Omron Sysmac Studio project BPP_17003_21Fev2018_13h32 (Sysmac Studio 1.21.1.6, StandardProject)

# Controller new_Controller_0: NJ101-1020 version 1.13
Units and slaves: Node10 : GX-JC06(IN,X2,X3) Main device (E001); Node11 : Inverter i550 Cabinet (E002); Node12 : Inverter i550 Cabinet (E003); Node13 : Inverter i550 Cabinet (E004); Node14 : Inverter i550 Cabinet (E005); Node15 : Inverter i550 Cabinet (E006); Node16 : Inverter i550 Cabinet (E007); Node21 : Inverter i550 Cabinet (E008); Node22 : Inverter i550 Cabinet (E009); Node23 : Inverter i550 Cabinet (E010); Node24 : Inverter i550 Cabinet (E011); Node25 : Inverter i550 Cabinet (E012); Node26 : Inverter i550 Cabinet (E013); Node30 : GX-JC06(X4,X5,X6) Sub-device (E014); Power Supply : NJ-Px3001; CPU : NJ101-1020; 0 [Unit 1] : CJ1W-ECT21 (J01); 1 [Unit 2] : CJ1W-EIP21 (J02); 2 : CJ1W-ID262 (J03); 3 : CJ1W-ID262 (J04); 4 : CJ1W-OD262 (J05); 5 : CJ1W-OD212 (J06)
Axis MC_Axis320M1, settings changed from default: AxisType=ServoType, UnitsConversion=EnumElement2, UnitsNumerator=8388608, UnitsDenominator=120, MaxVelocity=1000, StartVelocity=1000, MaxJogVelocity=100, MaxAcceleration=10, MaxDeceleration=10, WarningTorqueLimitPositive=90, WarningTorqueLimitNegative=90, HomingMode=BackupAndPressingTime, StartDirection=NegativeDirection, HomingVelocity=50, HomingApproachVelocity=10, HomingAcceleration=10, CompensationVelocity=10, EncoderTypes=Abs
Task PrimaryTask (priority 4, period or condition 2000): Programa

TYPE DataMotor : STRUCT
    Auto : BOOL;  (* Equipamento em Automatico *)
    Alarm : BOOL;  (* Equipamento em Alarme *)
    FcaFwd : BOOL;  (* Comando automatico Avanço *)
    FcaRev : BOOL;  (* Comando automatico Recuo *)
    FeFwd : BOOL;  (* Encravamento Avanço - Não pode Executar *)
    FeRev : BOOL;  (* Encravamento Recuo - Não pode Executar *)
    OutFwd : BOOL;  (* Output Avançar *)
    OutRev : BOOL;  (* Output Recuar *)
    FcaVel1 : BOOL;  (* Comando automatico velocidade 1 *)
    FcaVel2 : BOOL;  (* Comando automatico velocidade 2 *)
    OutVel1 : BOOL;  (* Output velocidade 1 *)
    OutVel2 : BOOL;  (* Output velocidade 2 *)
    JOGFwd : BOOL;  (* Jog Avanço *)
    JOGRev : BOOL;  (* Jog Recuo *)
    ManualLockIn : BOOL;  (* Lock infeed *)
    ManualLockOut : BOOL;  (* Lock Outfeed *)
    SetVel : INT;  (* Velocidade *)
    SetAcc : UINT;  (* Aceleração *)
    SetDec : UINT;  (* Desaceleração *)
END_STRUCT END_TYPE
TYPE Grafcet510M1 : STRUCT
    Step1 : BOOL;  (* Inicio *)
    Step2 : BOOL;  (* Procura Produto *)
    Step3 : BOOL;  (* Posiciona em 510YS2 *)
    Step4 : BOOL;  (* Produto Pronto a Entregar *)
    Step5 : BOOL;  (* A entregar produto *)
    Step6 : BOOL;  (* Produto Entregue *)
    Step7 : BOOL;
    Step8 : BOOL;
    Step9 : BOOL;
    Step10 : BOOL;  (* Pronto a receber *)
    Step11 : BOOL;  (* A receber Produto *)
    Step12 : BOOL;
    Step13 : BOOL;
    Step14 : BOOL;
    Step15 : BOOL;
    Step16 : BOOL;
    Step17 : BOOL;
    Step18 : BOOL;
    Step19 : BOOL;
    Step20 : BOOL;  (* Em Alarme - Necessario Retirar Produto Manual *)
    Step21 : BOOL;
    Step22 : BOOL;
    Step23 : BOOL;
    Step24 : BOOL;
    Step25 : BOOL;
    Step26 : BOOL;
    Step27 : BOOL;
    Step28 : BOOL;
    Step29 : BOOL;
    Step30 : BOOL;
    Step31 : BOOL;
    Step32 : BOOL;
END_STRUCT END_TYPE
TYPE Grafcet520M1 : STRUCT
    Step1 : BOOL;  (* Inicio *)
    Step2 : BOOL;  (* Procura Produto *)
    Step3 : BOOL;  (* Posiciona em 520YS1 *)
    Step4 : BOOL;  (* Produto Pronto a Entregar *)
    Step5 : BOOL;  (* A entregar produto *)
    Step6 : BOOL;
    Step7 : BOOL;
    Step8 : BOOL;
    Step9 : BOOL;
    Step10 : BOOL;  (* Pronto a receber *)
    Step11 : BOOL;  (* A receber Produto *)
    Step12 : BOOL;
    Step13 : BOOL;
    Step14 : BOOL;
    Step15 : BOOL;
    Step16 : BOOL;
    Step17 : BOOL;
    Step18 : BOOL;
    Step19 : BOOL;
    Step20 : BOOL;  (* Em Alarme - Necessario Retirar Produto Manual *)
    Step21 : BOOL;
    Step22 : BOOL;
    Step23 : BOOL;
    Step24 : BOOL;
    Step25 : BOOL;
    Step26 : BOOL;
    Step27 : BOOL;
    Step28 : BOOL;
    Step29 : BOOL;
    Step30 : BOOL;
    Step31 : BOOL;
    Step32 : BOOL;
END_STRUCT END_TYPE
TYPE Grafcet530M1 : STRUCT
    Step1 : BOOL;  (* Inicio *)
    Step2 : BOOL;  (* Procura Produto *)
    Step3 : BOOL;
    Step4 : BOOL;  (* Produto Pronto a Entregar *)
    Step5 : BOOL;  (* A entregar produto *)
    Step6 : BOOL;
    Step7 : BOOL;  (* Pack Posicionado para Impressao - Ordem de Ciclo de Impressao e Colagem *)
    Step8 : BOOL;  (* Posiciona produto na saida *)
    Step9 : BOOL;
    Step10 : BOOL;  (* Pronto a receber *)
    Step11 : BOOL;  (* A receber Produto *)
    Step12 : BOOL;  (* Espera paragem para dar trigger *)
    Step13 : BOOL;  (* A ler codigos de barras - Dá Trigger *)
    Step14 : BOOL;  (* A ler codigos de barras - Espera Resultado do Leitor *)
    Step15 : BOOL;  (* A ler codigos de barras - Guarda Resultado do Leitor *)
    Step16 : BOOL;  (* Fim de Codigos de Barras - Valida se tem 10 *)
    Step17 : BOOL;  (* Pergunta PC se válido *)
    Step18 : BOOL;  (* Aguarda Resposta do PC *)
    Step19 : BOOL;  (* Resposta do PC Ok - Posiciona para impressora *)
    Step20 : BOOL;  (* Em Alarme - Necessario Retirar Produto Manual *)
    Step21 : BOOL;  (* Em Alarme - Timeout à espera da resposta do PC *)
    Step22 : BOOL;  (* Em Alarme - Milheiros Invalidos *)
    Step23 : BOOL;  (* Em Alarme - Demasiado tempo para impressao *)
    Step24 : BOOL;
    Step25 : BOOL;
    Step26 : BOOL;
    Step27 : BOOL;
    Step28 : BOOL;
    Step29 : BOOL;
    Step30 : BOOL;
    Step31 : BOOL;
    Step32 : BOOL;
END_STRUCT END_TYPE
TYPE Grafcet540M1 : STRUCT
    Step1 : BOOL;  (* Inicio *)
    Step2 : BOOL;  (* Procura Produto *)
    Step3 : BOOL;  (* Indexa em 540YS1 *)
    Step4 : BOOL;  (* Posiciona no tapete em 540M2 *)
    Step5 : BOOL;  (* Procura em 540M1 *)
    Step6 : BOOL;  (* Pronto a Enviar *)
    Step7 : BOOL;  (* A enviar *)
    Step8 : BOOL;
    Step9 : BOOL;
    Step10 : BOOL;  (* Pronto a receber *)
    Step11 : BOOL;  (* A receber Produto *)
    Step12 : BOOL;
    Step13 : BOOL;
    Step14 : BOOL;
    Step15 : BOOL;
    Step16 : BOOL;
    Step17 : BOOL;
    Step18 : BOOL;
    Step19 : BOOL;
    Step20 : BOOL;  (* Em Alarme - Necessario Retirar Produto Manual *)
    Step21 : BOOL;
    Step22 : BOOL;
    Step23 : BOOL;
    Step24 : BOOL;
    Step25 : BOOL;
    Step26 : BOOL;
    Step27 : BOOL;
    Step28 : BOOL;
    Step29 : BOOL;
    Step30 : BOOL;
    Step31 : BOOL;
    Step32 : BOOL;
END_STRUCT END_TYPE
TYPE Grafcet6X0M1_Transport : STRUCT
    Step1 : BOOL;  (* Inicio *)
    Step2 : BOOL;  (* Procura Produto *)
    Step3 : BOOL;  (* Posiciona junto à saída *)
    Step4 : BOOL;  (* Pronto a Enviar *)
    Step5 : BOOL;  (* A enviar *)
    Step6 : BOOL;
    Step7 : BOOL;
    Step8 : BOOL;
    Step9 : BOOL;
    Step10 : BOOL;  (* Pronto a receber *)
    Step11 : BOOL;  (* A receber Produto *)
    Step12 : BOOL;
    Step13 : BOOL;
    Step14 : BOOL;
    Step15 : BOOL;
    Step16 : BOOL;
    Step17 : BOOL;
    Step18 : BOOL;
    Step19 : BOOL;
    Step20 : BOOL;  (* Em Alarme - Necessario Retirar Produto Manual *)
    Step21 : BOOL;
    Step22 : BOOL;
    Step23 : BOOL;
    Step24 : BOOL;
    Step25 : BOOL;
    Step26 : BOOL;
    Step27 : BOOL;
    Step28 : BOOL;
    Step29 : BOOL;
    Step30 : BOOL;
    Step31 : BOOL;
    Step32 : BOOL;
END_STRUCT END_TYPE
TYPE Grafcet6X0M1_Transport_Com2Transfer : STRUCT
    Step1 : BOOL;  (* Inicio *)
    Step2 : BOOL;  (* Procura Produto *)
    Step3 : BOOL;  (* Posiciona junto à saída *)
    Step4 : BOOL;  (* Pronto a Enviar *)
    Step5 : BOOL;  (* A enviar *)
    Step6 : BOOL;  (* Posiciona junto à 1.a Transfer *)
    Step7 : BOOL;  (* Descarrega para a 1.a Transfer *)
    Step8 : BOOL;  (* Posiciona junto à 2.a Transfer *)
    Step9 : BOOL;  (* Descarrega para a 2.a Transfer *)
    Step10 : BOOL;  (* Pronto a receber *)
    Step11 : BOOL;  (* A receber Produto *)
    Step12 : BOOL;
    Step13 : BOOL;
    Step14 : BOOL;
    Step15 : BOOL;
    Step16 : BOOL;
    Step17 : BOOL;
    Step18 : BOOL;
    Step19 : BOOL;
    Step20 : BOOL;  (* Em Alarme - Necessario Retirar Produto Manual *)
    Step21 : BOOL;
    Step22 : BOOL;
    Step23 : BOOL;
    Step24 : BOOL;
    Step25 : BOOL;
    Step26 : BOOL;
    Step27 : BOOL;
    Step28 : BOOL;
    Step29 : BOOL;
    Step30 : BOOL;
    Step31 : BOOL;
    Step32 : BOOL;
END_STRUCT END_TYPE
TYPE Grafcet550U1 : STRUCT
    Step1 : BOOL;  (* Inicio *)
    Step2 : BOOL;  (* Verifica Condicoes de Funcionamento *)
    Step3 : BOOL;  (* Aguarda produto posicionado *)
    Step4 : BOOL;  (* Prepara Sistema para Ordem de Impressao *)
    Step5 : BOOL;  (* Da Ordem de Impressao *)
    Step6 : BOOL;  (* Espera Fim de Ordem de Impressao *)
    Step7 : BOOL;  (* Espera Fim de Rebobinar *)
    Step8 : BOOL;  (* Desliga Sopro *)
    Step9 : BOOL;  (* Avanca Pneumatico *)
    Step10 : BOOL;  (* Desliga Vacuo *)
    Step11 : BOOL;  (* Recolhe Pneumatico *)
    Step12 : BOOL;  (* Impressao Ok *)
    Step13 : BOOL;
    Step14 : BOOL;
    Step15 : BOOL;
    Step16 : BOOL;
    Step17 : BOOL;
    Step18 : BOOL;
    Step19 : BOOL;
    Step20 : BOOL;  (* Alarme: Cilindro não recolhe *)
    Step21 : BOOL;  (* Alarme: Demasiado tempo em impressao *)
    Step22 : BOOL;  (* Alarme: Demasiado tempo a rebobinar *)
    Step23 : BOOL;  (* Alarme - Erro em impressao pelo PC *)
    Step24 : BOOL;
    Step25 : BOOL;
    Step26 : BOOL;
    Step27 : BOOL;
    Step28 : BOOL;
    Step29 : BOOL;
    Step30 : BOOL;
    Step31 : BOOL;
    Step32 : BOOL;
END_STRUCT END_TYPE
TYPE Position : STRUCT
    Position0 : LREAL;  (* Posição 0 *)
    Position1 : LREAL;  (* Posição 1 *)
    Position2 : LREAL;  (* Posição 2 *)
    GoToPos0 : BOOL;  (* Ir para posição 0 *)
    GoToPos1 : BOOL;  (* Ir para posição 1 *)
    GoToPos2 : BOOL;  (* Ir para posição 2 *)
    InPos0 : BOOL;  (* Em posição 0 *)
    InPos1 : BOOL;  (* Em posição 1 *)
    InPos2 : BOOL;  (* Em posição 2 *)
END_STRUCT END_TYPE
TYPE DataServo : STRUCT
    PowerOn : BOOL;  (* Alimentação Ligada *)
    Ready : BOOL;  (* Servo/Drive Ready - Sem Erros *)
    Auto : BOOL;  (* Servo em Automatico *)
    Free : BOOL;  (* Servo Disponível *)
    ExecHome : BOOL;  (* Executa Home Position *)
    Homed : BOOL;  (* Home Done *)
    JogFwd : BOOL;  (* Jog Fwd *)
    JogRev : BOOL;  (* Jog Rev *)
    JogFwdAux : BOOL;  (* Jog Fwd - Auxiliar *)
    JogRevAux : BOOL;  (* Jog Rev - Auxiliar *)
    Speed : LREAL;
    Accel : LREAL;
    Deccel : LREAL;
    Jerk : LREAL;
END_STRUCT END_TYPE
TYPE Alarme : STRUCT
    Alarme1 : BOOL;
    Alarme2 : BOOL;
    Alarme3 : BOOL;
    Alarme4 : BOOL;
    Alarme5 : BOOL;
    Alarme6 : BOOL;
    Alarme7 : BOOL;
    Alarme8 : BOOL;
    Alarme9 : BOOL;
    Alarme10 : BOOL;
    Alarme11 : BOOL;
    Alarme12 : BOOL;
    Alarme13 : BOOL;
    Alarme14 : BOOL;
    Alarme15 : BOOL;
    Alarme16 : BOOL;
    Alarme17 : BOOL;
    Alarme18 : BOOL;
    Alarme19 : BOOL;
    Alarme20 : BOOL;
END_STRUCT END_TYPE
TYPE AlarmeGeralLinha : STRUCT
    Alarme1 : BOOL;  (* Emergência *)
    Alarme2 : BOOL;  (* Falha Ar Comprimido *)
    Alarme3 : BOOL;  (* Falha Fonte 24Vdc *)
    Alarme4 : BOOL;
    Alarme5 : BOOL;
    Alarme6 : BOOL;
    Alarme7 : BOOL;
    Alarme8 : BOOL;
    Alarme9 : BOOL;
    Alarme10 : BOOL;
    Alarme11 : BOOL;
    Alarme12 : BOOL;
    Alarme13 : BOOL;
    Alarme14 : BOOL;
    Alarme15 : BOOL;
    Alarme16 : BOOL;
    Alarme17 : BOOL;
    Alarme18 : BOOL;
    Alarme19 : BOOL;
    Alarme20 : BOOL;
END_STRUCT END_TYPE
TYPE DataValve : STRUCT
    Auto : BOOL;  (* Equipamento em Automatico *)
    Alarm : BOOL;  (* Equipamento em Alarme *)
    FcaFwd : BOOL;  (* Comando automatico Avanço *)
    FcaRev : BOOL;  (* Comando automatico Recuo *)
    FeFwd : BOOL;  (* Encravamento Avanço - Não pode Executar *)
    FeRev : BOOL;  (* Encravamento Recuo - Não pode Executar *)
    OutFwd : BOOL;  (* Output Avançar *)
    OutRev : BOOL;  (* Output Recuar *)
    JOGFwd : BOOL;  (* Jog Avanço *)
    JOGRev : BOOL;  (* Jog Recuo *)
END_STRUCT END_TYPE
TYPE AlarmeGeralEquipamento : STRUCT
    Alarme1 : BOOL;  (* Alarme Defeito *)
    Alarme2 : BOOL;  (* Aviso Alarme - Necessario Stop *)
    Alarme3 : BOOL;  (* Alarme Motion *)
    Alarme4 : BOOL;  (* Alarme Segurança *)
    Alarme5 : BOOL;  (* Alarme Estado *)
    Alarme6 : BOOL;  (* Alarme Grafcet Equipamento *)
    Alarme7 : BOOL;  (* Alarme Externo *)
    Alarme8 : BOOL;
    Alarme9 : BOOL;
    Alarme10 : BOOL;
    Alarme11 : BOOL;
    Alarme12 : BOOL;
    Alarme13 : BOOL;
    Alarme14 : BOOL;
    Alarme15 : BOOL;
    Alarme16 : BOOL;
    Alarme17 : BOOL;
    Alarme18 : BOOL;
    Alarme19 : BOOL;
    Alarme20 : BOOL;
END_STRUCT END_TYPE
TYPE Event : STRUCT
    Event1 : BOOL;
    Event2 : BOOL;
    Event3 : BOOL;
    Event4 : BOOL;
    Event5 : BOOL;
    Event6 : BOOL;
    Event7 : BOOL;
    Event8 : BOOL;
    Event9 : BOOL;
    Event10 : BOOL;
    Event11 : BOOL;
    Event12 : BOOL;
    Event13 : BOOL;
    Event14 : BOOL;
    Event15 : BOOL;
    Event16 : BOOL;
    Event17 : BOOL;
    Event18 : BOOL;
    Event19 : BOOL;
    Event20 : BOOL;
END_STRUCT END_TYPE
TYPE Grafcet : STRUCT
    Step1 : BOOL;
    Step2 : BOOL;
    Step3 : BOOL;
    Step4 : BOOL;
    Step5 : BOOL;
    Step6 : BOOL;
    Step7 : BOOL;
    Step8 : BOOL;
    Step9 : BOOL;
    Step10 : BOOL;
    Step11 : BOOL;
    Step12 : BOOL;
    Step13 : BOOL;
    Step14 : BOOL;
    Step15 : BOOL;
    Step16 : BOOL;
    Step17 : BOOL;
    Step18 : BOOL;
    Step19 : BOOL;
    Step20 : BOOL;
END_STRUCT END_TYPE
TYPE Grafcet111U1 : STRUCT
    Step1 : BOOL;  (* Inicio *)
    Step2 : BOOL;  (* Limpa Variaveis *)
    Step3 : BOOL;  (* Variaveis Limpas *)
    Step4 : BOOL;  (* Código Validado *)
    Step5 : BOOL;  (* Verifica Ano *)
    Step6 : BOOL;  (* Verifica Dia Juliano *)
    Step7 : BOOL;  (* Verifica Máquina e atribui ID *)
    Step8 : BOOL;  (* Verifica se tem destino Atribuido *)
    Step9 : BOOL;  (* Código Validado *)
    Step10 : BOOL;  (* Reinicia Grafecet *)
    Step11 : BOOL;
    Step12 : BOOL;
    Step13 : BOOL;
    Step14 : BOOL;
    Step15 : BOOL;
    Step16 : BOOL;
    Step17 : BOOL;
    Step18 : BOOL;
    Step19 : BOOL;
    Step20 : BOOL;
END_STRUCT END_TYPE
TYPE Grafcet250U1 : STRUCT
    Step1 : BOOL;  (* Inicio *)
    Step2 : BOOL;  (* Limpa Variaveis *)
    Step3 : BOOL;  (* Variaveis Limpas *)
    Step4 : BOOL;  (* Código Validado *)
    Step5 : BOOL;  (* Escreveu primeiro ID *)
    Step6 : BOOL;  (* Verificou ID restantes *)
    Step7 : BOOL;  (* Código Validado *)
    Step8 : BOOL;  (* Reinicia Grafecet *)
    Step9 : BOOL;
    Step10 : BOOL;
    Step11 : BOOL;
    Step12 : BOOL;
    Step13 : BOOL;
    Step14 : BOOL;
    Step15 : BOOL;
    Step16 : BOOL;
    Step17 : BOOL;
    Step18 : BOOL;
    Step19 : BOOL;
    Step20 : BOOL;
END_STRUCT END_TYPE
TYPE DataProd : STRUCT
    Machine : UINT;  (* Nr Máquina de Escolha *)
    NotaType : UINT;  (* Tipo de Nota *)
    QtdActual : UINT;  (* Quantidade de Milheiros no Transportador *)
    ProdID : UINT;  (* ID do Produto *)
END_STRUCT END_TYPE
TYPE DataBuffer : STRUCT
    QtdTotal : UINT;  (* Quantidade Total de Milheiros no Buffer *)
    WaitTime : UINT;  (* Tempo de Espera para Descarga *)
    PedeDescargaToReject : BOOL;  (* Pedido de descarga para Rejeitados *)
    DescargaAtribuidaToRobot : BOOL;  (* Descarga Atribuida para Robot *)
    DescargaAtribuidaToReject : BOOL;  (* Descarga Atribuida para Rejeitados *)
END_STRUCT END_TYPE
TYPE GrafcetEmpurrador : STRUCT
    Step1 : BOOL;  (* Inicio *)
    Step2 : BOOL;  (* Empurrador Recuado *)
    Step3 : BOOL;  (* Recebe ordem para avançar *)
    Step4 : BOOL;  (* Empurrador Avançado *)
    Step5 : BOOL;  (* Recebe ordem para recuar *)
    Step6 : BOOL;
    Step7 : BOOL;
    Step8 : BOOL;
    Step9 : BOOL;
    Step10 : BOOL;
    Step11 : BOOL;
    Step12 : BOOL;
    Step13 : BOOL;
    Step14 : BOOL;
    Step15 : BOOL;
    Step16 : BOOL;
    Step17 : BOOL;
    Step18 : BOOL;
    Step19 : BOOL;
    Step20 : BOOL;
END_STRUCT END_TYPE
TYPE DataTransport : STRUCT
    ModeRev : BOOL;  (* (=0 Fwd ; =1 Rev) *)
    ModeBuffer : BOOL;  (* (=0 Não Acumula Produto ; =1 Acumula Produto) *)
    ReadyToSend : BOOL;  (* Com produto para Enviar *)
    ReadyToReceive : BOOL;  (* Pronto a receber *)
    RollersRunningIn : BOOL;  (* Rolos a andar Infeed *)
    RollersRunningOut : BOOL;  (* Rolos a andar Outfeed *)
    ReceiveEnd : BOOL;
    InfeedStart : BOOL;
    InfeedGoTo : BOOL;
    InfeedFwd : BOOL;
    InfeedRev : BOOL;
    InfeedInTrip : BOOL;
    InfeedTimeOut : BOOL;  (* Time Out *)
    InfeedTimeOutRev : BOOL;  (* Time Out *)
    OutfeedStart : BOOL;
    OutfeedGoTo : BOOL;
    OutfeedFwd : BOOL;
    OutfeedRev : BOOL;
    OutfeedInTrip : BOOL;
    OutfeedInTripRev : BOOL;
    OutfeedAjust : BOOL;
    OutfeedTimeOut : BOOL;  (* Time Out *)
    OutfeedTimeOutRev : BOOL;  (* Time Out *)
    TimeOutSet : UINT;  (* Tempo de espera para TimeOut *)
    TimeOut : BOOL;  (* Time Out *)
    Busy : BOOL;  (* Ocupado *)
    Full : BOOL;  (* Transportador Cheio *)
    Free : BOOL;  (* Livre - Sem movimentos *)
END_STRUCT END_TYPE
TYPE GrafcetBatente : STRUCT
    Step1 : BOOL;  (* Inicio - Verifica se tem produto *)
    Step2 : BOOL;  (* Batente Livre *)
    Step3 : BOOL;  (* Batente em cima *)
    Step4 : BOOL;  (* Batente com produto para entregar *)
    Step5 : BOOL;  (* Foi pedido produto *)
    Step6 : BOOL;  (* Produto a ser entregue *)
    Step7 : BOOL;  (* Entregou produto *)
    Step8 : BOOL;
    Step9 : BOOL;
    Step10 : BOOL;
    Step11 : BOOL;
    Step12 : BOOL;
    Step13 : BOOL;
    Step14 : BOOL;
    Step15 : BOOL;
    Step16 : BOOL;
    Step17 : BOOL;
    Step18 : BOOL;
    Step19 : BOOL;
    Step20 : BOOL;
END_STRUCT END_TYPE
TYPE GrafcetAcumula : STRUCT
    Step1 : BOOL;  (* Inicio *)
    Step2 : BOOL;  (* Procura Produto *)
    Step3 : BOOL;  (* Não Encontrou Produto Transportador Vazio *)
    Step4 : BOOL;  (* Encontrou Produto *)
    Step5 : BOOL;  (* Transportador Parado *)
    Step6 : BOOL;  (* Pronto a receber *)
    Step7 : BOOL;  (* A receber *)
    Step8 : BOOL;  (* Produto a entrar *)
    Step9 : BOOL;  (* Produto carregado *)
    Step10 : BOOL;  (* Produto posicionado *)
    Step11 : BOOL;  (* Produto incrementado *)
    Step12 : BOOL;  (* Transportador Parado após incrementar *)
    Step13 : BOOL;  (* Carga Incompleta *)
    Step14 : BOOL;  (* Carga Completa *)
    Step15 : BOOL;  (* Avanço para saida *)
    Step16 : BOOL;  (* Chegou produto à fotocelula de saida *)
    Step17 : BOOL;  (* Espera descarga *)
    Step18 : BOOL;  (* Descarga atribuida *)
    Step19 : BOOL;  (* Em Descarga *)
    Step20 : BOOL;  (* Finalizou descarga *)
    Step21 : BOOL;  (* Avança para saida - Rejeitados *)
    Step22 : BOOL;  (* Chegou produto à fotocelula de saida - Rejeitados *)
    Step23 : BOOL;  (* Espera descarga - Rejeitados *)
    Step24 : BOOL;  (* Descarga atribuida - Rejeitados *)
    Step25 : BOOL;  (* Em Descarga - Rejeitados *)
    Step26 : BOOL;  (* Finalizou descarga - Rejeitados *)
    Step27 : BOOL;
    Step28 : BOOL;
    Step29 : BOOL;
    Step30 : BOOL;
    Step31 : BOOL;
    Step32 : BOOL;
END_STRUCT END_TYPE
TYPE Grafcet230M1 : STRUCT
    Step1 : BOOL;  (* Inicio *)
    Step2 : BOOL;  (* Procura Produto *)
    Step3 : BOOL;  (* Não Encontrou Produto Transportador Vazio *)
    Step4 : BOOL;  (* Encontrou Produto *)
    Step5 : BOOL;  (* Transportador Parado *)
    Step6 : BOOL;  (* Pronto a receber *)
    Step7 : BOOL;  (* A receber para Robot *)
    Step8 : BOOL;  (* Produto a entrar *)
    Step9 : BOOL;  (* Produto na fotocelula de saida *)
    Step10 : BOOL;  (* Em descarga *)
    Step11 : BOOL;  (* Produto decrementado *)
    Step12 : BOOL;  (* Descarga Incompleta *)
    Step13 : BOOL;  (* Descarga Completa *)
    Step14 : BOOL;  (* Descarga Finalizada *)
    Step15 : BOOL;  (* A receber para Rejeitados *)
    Step16 : BOOL;  (* Produto a entrar para rejeitados *)
    Step17 : BOOL;  (* Descarga Rejeitados completa *)
    Step18 : BOOL;
    Step19 : BOOL;
    Step20 : BOOL;
    Step21 : BOOL;
    Step22 : BOOL;
    Step23 : BOOL;
    Step24 : BOOL;
    Step25 : BOOL;
    Step26 : BOOL;
    Step27 : BOOL;
    Step28 : BOOL;
    Step29 : BOOL;
    Step30 : BOOL;
    Step31 : BOOL;
    Step32 : BOOL;
END_STRUCT END_TYPE
TYPE Grafcet240M1 : STRUCT
    Step1 : BOOL;  (* Inicio *)
    Step2 : BOOL;  (* Procura Produto *)
    Step3 : BOOL;  (* Não Encontrou Produto Transportador Vazio *)
    Step4 : BOOL;  (* Encontrou Produto *)
    Step5 : BOOL;  (* Transportador Parado *)
    Step6 : BOOL;  (* Pronto a receber *)
    Step7 : BOOL;  (* A receber *)
    Step8 : BOOL;  (* Produto a entrar ou procura do próximo produto *)
    Step9 : BOOL;  (* Produto na fotocelula de saida *)
    Step10 : BOOL;  (* Em descarga *)
    Step11 : BOOL;  (* Produto saiu do transportador *)
    Step12 : BOOL;  (* Descarga Completa *)
    Step13 : BOOL;  (* Descarga Finalizada *)
    Step14 : BOOL;
    Step15 : BOOL;
    Step16 : BOOL;
    Step17 : BOOL;
    Step18 : BOOL;
    Step19 : BOOL;
    Step20 : BOOL;
    Step21 : BOOL;
    Step22 : BOOL;
    Step23 : BOOL;
    Step24 : BOOL;
    Step25 : BOOL;
    Step26 : BOOL;
    Step27 : BOOL;
    Step28 : BOOL;
    Step29 : BOOL;
    Step30 : BOOL;
    Step31 : BOOL;
    Step32 : BOOL;
END_STRUCT END_TYPE
TYPE Grafcet250M1 : STRUCT
    Step1 : BOOL;  (* Inicio *)
    Step2 : BOOL;  (* Procura Produto *)
    Step3 : BOOL;  (* Não Encontrou Produto Transportador Vazio *)
    Step4 : BOOL;  (* Encontrou Produto *)
    Step5 : BOOL;  (* Transportador Parado *)
    Step6 : BOOL;  (* Pronto a receber *)
    Step7 : BOOL;  (* A receber *)
    Step8 : BOOL;  (* Produto a entrar *)
    Step9 : BOOL;  (* Produto carregado *)
    Step10 : BOOL;  (* Produto na fotocelula do LCB *)
    Step11 : BOOL;  (* A posicionar produto na Fotocelula LCB *)
    Step12 : BOOL;  (* Produto posicionado *)
    Step13 : BOOL;  (* Ordem de Leitura de Código Barras *)
    Step14 : BOOL;  (* Espera Leitura Código de Barras *)
    Step15 : BOOL;  (* Verifica Código OK ou NOK *)
    Step16 : BOOL;  (* Código OK - Gera ID *)
    Step17 : BOOL;  (* Código NOK - Coloca ID #0 *)
    Step18 : BOOL;  (* Avança para Empurrador *)
    Step19 : BOOL;  (* Produto a Indexar *)
    Step20 : BOOL;  (* Produto Indexado no Empurrador *)
    Step21 : BOOL;  (* Produto Pronto a Entregar *)
    Step22 : BOOL;  (* Produto a entregar *)
    Step23 : BOOL;  (* Produto Entregue - Empurrador Frontal *)
    Step24 : BOOL;  (* Produto Entregue - Avanço Empurrador Lateral *)
    Step25 : BOOL;  (* Produto Entregue - Pronto a pegar *)
    Step26 : BOOL;  (* Produto Decrementado *)
    Step27 : BOOL;  (* Entrega Incompleta *)
    Step28 : BOOL;  (* Entrega Completa *)
    Step29 : BOOL;  (* Entrega Finalizada *)
    Step30 : BOOL;
    Step31 : BOOL;
    Step32 : BOOL;
END_STRUCT END_TYPE
TYPE Grafcet310M1 : STRUCT
    Step1 : BOOL;  (* Inicio *)
    Step2 : BOOL;  (* Procura Produto *)
    Step3 : BOOL;  (* Não Encontrou Produto Transportador Vazio *)
    Step4 : BOOL;  (* Encontrou Produto *)
    Step5 : BOOL;  (* Transportador Parado *)
    Step6 : BOOL;  (* Pronto a receber *)
    Step7 : BOOL;  (* Robot iniciou entrega de produto *)
    Step8 : BOOL;  (* Robot Finalizou entrega de produto *)
    Step9 : BOOL;  (* Robot saiu da mesa após finalizar entrega de produto *)
    Step10 : BOOL;  (* Efetua pré indixação *)
    Step11 : BOOL;  (* Sobe mesa *)
    Step12 : BOOL;  (* Indexa milheiros lateralmente *)
    Step13 : BOOL;  (* Milheiros Indexados *)
    Step14 : BOOL;  (* Abre indexador *)
    Step15 : BOOL;  (* Indexa Milheiros à Retaguarda *)
    Step16 : BOOL;  (* A indexar Milheiros *)
    Step17 : BOOL;  (* Produto Indexado no Batente *)
    Step18 : BOOL;  (* Pronto a entregar à Ulma *)
    Step19 : BOOL;  (* Produto a entregar *)
    Step20 : BOOL;  (* Produto chegou à fotocelula de saida *)
    Step21 : BOOL;  (* Produto a entrar na ULMA *)
    Step22 : BOOL;  (* Esvazia Transportador *)
    Step23 : BOOL;  (* Descarga Finalizada *)
    Step24 : BOOL;
    Step25 : BOOL;
    Step26 : BOOL;
    Step27 : BOOL;
    Step28 : BOOL;
    Step29 : BOOL;
    Step30 : BOOL;
    Step31 : BOOL;
    Step32 : BOOL;
END_STRUCT END_TYPE
TYPE In_EIPMulticontrol : STRUCT
    Input1 : ARRAY[0..23] OF BOOL;
    Speed : ARRAY[0..5] OF BYTE;
    MotorCurrent1 : WORD;
    MotorCurrent2 : WORD;
    MotorCurrent3 : WORD;
    MotorCurrent4 : WORD;
    Voltage1 : WORD;
    Voltage2 : WORD;
    Temperature : WORD;
    SystemUpTime : WORD;
    Input2 : ARRAY[0..9] OF BYTE;
END_STRUCT END_TYPE
TYPE Out_EIPMulticontrol : STRUCT
    Speed : ARRAY[0..4] OF BYTE;
    Output1 : ARRAY[0..23] OF BOOL;
END_STRUCT END_TYPE
TYPE Interroll : STRUCT
    Sensor : BOOL;
    Error : BOOL;
    Run : BOOL;
    Free : BOOL;  (* Livre sem movimentos *)
    RdyToSend : BOOL;  (* Pronto a enviar *)
    RdyToRcv : BOOL;  (* Pronto a receber *)
    InfeedStart : BOOL;
    InfeedFwd : BOOL;
    InfeedInTrip : BOOL;
    InfeedGoTo : BOOL;
    OutfeedStart : BOOL;
    OutfeedFwd : BOOL;
    OutfeedInTrip : BOOL;
    OutfeedGoTo : BOOL;
    Speed_Target : INT;
END_STRUCT END_TYPE
TYPE Grafcet111M1 : STRUCT
    Step1 : BOOL;  (* Inicio *)
    Step2 : BOOL;  (* Procura Produto *)
    Step3 : BOOL;  (* Não Encontrou Produto Transportador Vazio *)
    Step4 : BOOL;  (* Encontrou Produto *)
    Step5 : BOOL;  (* Transportador Parado *)
    Step6 : BOOL;  (* Pronto a receber *)
    Step7 : BOOL;  (* A receber *)
    Step8 : BOOL;  (* Produto a entrar *)
    Step9 : BOOL;  (* Produto carregado *)
    Step10 : BOOL;  (* Produto na fotocelula LCB *)
    Step11 : BOOL;  (* A posicionar produto na Fotocelula LCB *)
    Step12 : BOOL;  (* Produto posicionado *)
    Step13 : BOOL;  (* Ordem de Leitura de Código Barras *)
    Step14 : BOOL;  (* Espera Leitura Código de Barras *)
    Step15 : BOOL;  (* Verifica Código OK ou NOK *)
    Step16 : BOOL;  (* Código OK - Gera ID *)
    Step17 : BOOL;  (* Código NOK - Coloca ID #0 *)
    Step18 : BOOL;  (* Avança para Empurrador *)
    Step19 : BOOL;  (* Produto na Fotocelula do empurrador *)
    Step20 : BOOL;  (* Produto a Indexar *)
    Step21 : BOOL;  (* Produto Indexado no Empurrador *)
    Step22 : BOOL;  (* Produto Pronto a Entregar *)
    Step23 : BOOL;  (* Produto a entregar *)
    Step24 : BOOL;  (* Produto Entregue *)
    Step25 : BOOL;
    Step26 : BOOL;
    Step27 : BOOL;
    Step28 : BOOL;
    Step29 : BOOL;
    Step30 : BOOL;
    Step31 : BOOL;
    Step32 : BOOL;
END_STRUCT END_TYPE
TYPE Grafcet120M1 : STRUCT
    Step1 : BOOL;  (* Inicio *)
    Step2 : BOOL;  (* Procura Produto *)
    Step3 : BOOL;  (* Transportador Vazio *)
    Step4 : BOOL;  (* Transportador Parado *)
    Step5 : BOOL;  (* Pronto a receber *)
    Step6 : BOOL;  (* A receber *)
    Step7 : BOOL;  (* Produto a entrar *)
    Step8 : BOOL;  (* Produto carregado *)
    Step9 : BOOL;  (* Produto em circulação *)
    Step10 : BOOL;  (* Produto para Buffer 1 *)
    Step11 : BOOL;  (* Produto a posicionar para Buffer 1 *)
    Step12 : BOOL;  (* Produto posicionado para Buffer 1 *)
    Step13 : BOOL;  (* Produto para Buffer 2 *)
    Step14 : BOOL;  (* Produto a posicionar para Buffer 2 *)
    Step15 : BOOL;  (* Produto posicionado para Buffer 2 *)
    Step16 : BOOL;  (* Produto para Buffer 3 *)
    Step17 : BOOL;  (* Produto a posicionar para Buffer 3 *)
    Step18 : BOOL;  (* Produto posicionado para Buffer 3 *)
    Step19 : BOOL;  (* Produto saiu do transportador *)
    Step20 : BOOL;  (* Produto entregue no Buffer correspondente *)
    Step21 : BOOL;  (* Transportador vazio *)
    Step22 : BOOL;
    Step23 : BOOL;
    Step24 : BOOL;
    Step25 : BOOL;
    Step26 : BOOL;
    Step27 : BOOL;
    Step28 : BOOL;
    Step29 : BOOL;
    Step30 : BOOL;
    Step31 : BOOL;
    Step32 : BOOL;
END_STRUCT END_TYPE
TYPE DataLCB : STRUCT
    NotaType : UINT;  (* Tipo de Nota *)
    Center : UINT;  (* Centro de Escolha *)
    MachineNr : UINT;  (* Numero de Máquina *)
    MilheiroNr : UINT;  (* Numero de Milheiro *)
    Year : UINT;  (* Ano *)
    ZeroDigit : UINT;  (* Valor Fixo Zero *)
    JulianDate : UINT;  (* Data Juliana *)
    CheckDigit : UINT;  (* Check Digit *)
    EAN13 : STRING[128];  (* Código Completo *)
    Busy : BOOL;  (* Ocupado a efetuar calculo *)
    CodeOK : BOOL;  (* Codigo Lido com Sucesso *)
    CodeNOK : BOOL;  (* Código Não lido *)
    Clear : BOOL;  (* Apagar Dados de leitura *)
END_STRUCT END_TYPE
TYPE SafetyIn_struct : STRUCT
    Watchdog : BOOL;  (* Watchdog (Pulse a 1seg) *)
    Botoneiras : BOOL;  (* Estado Actual das Botoneiras *)
    Porta : BOOL;  (* Estado Actual da Porta *)
    GeralOk : BOOL;  (* Safety Ok - Zona Geral *)
    Z300Ok : BOOL;  (* Safety Ok - Zona 300 *)
END_STRUCT END_TYPE
TYPE SafetyOut_struct : STRUCT
    Watchdog : BOOL;  (* Watchdog (Pulse a 1seg) *)
    TrincoAberturaPorta : BOOL;
    LedPedidoAberturaPorta : BOOL;
END_STRUCT END_TYPE

VAR_GLOBAL
    Pulse_1s : BOOL := False;  (* Pulse 1s *)
    Pulse_100ms : BOOL := False;  (* Pulse 100ms *)
    Pulse_2s : BOOL := False;  (* Pulse 2s *)
    Pulse_5s : BOOL := False;  (* Pulse 5s *)
    Pulse_10ms : BOOL := False;  (* Pulse 10ms *)
    Pulse_30s : BOOL := False;  (* Pulse 30s *)
END_VAR
VAR_GLOBAL RETAIN
    G_Robot : Grafcet;  (* Grafcet Equipamento *)
END_VAR
VAR_GLOBAL
    A_320M1 : AlarmeGeralEquipamento;
END_VAR
VAR_GLOBAL RETAIN
    G_111V : GrafcetEmpurrador;
END_VAR
VAR_GLOBAL
    StartRobot : BOOL;  (* 330 - Inicio de Automatico Externo do Robot; published *)
    Q_330V1 : BOOL;  (* 330V1 - Valvula Ferramenta Robot Abrir; at IOBus://rack#0/slot#4/Ch3_Out/Ch3_Out12 *)
    IFQ_330_DrivesOff : BOOL;  (* 330 - Robot Drives OFF; published *)
    IFQ_330_ConfMess : BOOL;  (* 330 - Robot ACK; published *)
    IFQ_330_DrivesOn : BOOL;  (* 330 - Robot Drives ON; published *)
    IFQ_330_ExtStart : BOOL;  (* 330 - Robot External Start; published *)
    IFQ_330_MoveEnable : BOOL;  (* 330 - Robot Move Enable; published *)
    IFQ_330_WatchDog : BOOL;  (* 330 - WatchDog; published *)
    I_300HS1 : BOOL;  (* 300HS1 - Botoneira de Start; at IOBus://rack#0/slot#3/Ch2_In/Ch2_In11 *)
    Zona300On : BOOL;  (* Zona 300 Ligada; published *)
    I_300HS2 : BOOL;  (* 300HS2 - Botoneira de Stop; at IOBus://rack#0/slot#3/Ch2_In/Ch2_In12 *)
    CondGerais300OK : BOOL;  (* Condições Gerais Zona 300 OK para funcionamento; published *)
    IFQ_330_RdytoPick : BOOL;  (* 330 - Ready to Pick From 250; published *)
    IFQ_330_RdytoPlace : BOOL;  (* 330 - Ready to Place to 310; published *)
    JulianDate : LINT;
    IFQ_330_Rst310 : BOOL;  (* 330 - Reset Zona 310 (Obriga Reset Robot); published *)
    IFQ_330_NewData : BOOL;  (* 330 - Novos Dados em 250; published *)
    IFQ_330_DataOK : BOOL;  (* 330 - Dados Validados; published *)
    A_110V : AlarmeGeralEquipamento;  (* published *)
    A_111V : AlarmeGeralEquipamento;  (* published *)
    A_121V : AlarmeGeralEquipamento;  (* published *)
    A_122V : AlarmeGeralEquipamento;  (* published *)
    A_123V : AlarmeGeralEquipamento;  (* published *)
    A_211V : AlarmeGeralEquipamento;  (* published *)
    A_212V : AlarmeGeralEquipamento;  (* published *)
    A_213V : AlarmeGeralEquipamento;  (* published *)
    A_251V : AlarmeGeralEquipamento;  (* published *)
    A_252V : AlarmeGeralEquipamento;  (* published *)
    A_321V : AlarmeGeralEquipamento;  (* published *)
    A_Geral : AlarmeGeralLinha;  (* published *)
    D_110V : DataValve;  (* Data Valve; published *)
    D_111V : DataValve;  (* Data Valve; published *)
    D_121V : DataValve;  (* Data Valve; published *)
    D_122V : DataValve;  (* Data Valve; published *)
    D_123V : DataValve;  (* Data Valve; published *)
    D_211V : DataValve;  (* Data Valve; published *)
    D_212V : DataValve;  (* Data Valve; published *)
    D_213V : DataValve;  (* Data Valve; published *)
    D_251V : DataValve;  (* Data Valve; published *)
    D_252V : DataValve;  (* Data Valve; published *)
    D_321V : DataValve;  (* Data Valve; published *)
    E_110V : Event;  (* Event; published *)
    E_111V : Event;  (* Event; published *)
    E_121V : Event;  (* Event; published *)
    E_122V : Event;  (* Event; published *)
    E_123V : Event;  (* Event; published *)
    E_211V : Event;  (* Event; published *)
    E_212V : Event;  (* Event; published *)
    E_213V : Event;  (* Event; published *)
    E_251V : Event;  (* Event; published *)
    E_252V : Event;  (* Event; published *)
    E_321V : Event;  (* Event; published *)
    IFI_330_WORD1 AT %200 : ARRAY[0..15] OF BOOL;
    IFQ_330_WORD1 AT %400 : ARRAY[0..15] OF BOOL;
    I_110YS1 : BOOL;  (* 110YS1 - Fotocelula Linha Cheia; at IOBus://rack#0/slot#2/Ch2_In/Ch2_In00 *)
    I_110YS2 : BOOL;  (* 110YS2 - Fotocelula Saida Transportador; at IOBus://rack#0/slot#2/Ch2_In/Ch2_In01 *)
    I_110XS1 : BOOL;  (* 110XS1 - Sensor Batente Saida em Cima; at IOBus://rack#0/slot#2/Ch2_In/Ch2_In02 *)
    I_110XS2 : BOOL;  (* 110XS2 - Sensor Batente Saida em Baixo; at IOBus://rack#0/slot#2/Ch2_In/Ch2_In03 *)
    I_111U1OK : BOOL;  (* 111U1OK - Output Leitura OK (Output 1); at IOBus://rack#0/slot#2/Ch2_In/Ch2_In04 *)
    I_111YS1 : BOOL;  (* 111YS1 - Fotocelula Posição Leitura Codigo Barras; at IOBus://rack#0/slot#2/Ch2_In/Ch2_In06 *)
    I_111YS2 : BOOL;  (* 111YS2 - Fotocelula Milheiro Indexado; at IOBus://rack#0/slot#2/Ch2_In/Ch2_In07 *)
    I_111XS1 : BOOL;  (* 111XS1 - Sensor Empurrador Lateral Avancado; at IOBus://rack#0/slot#2/Ch2_In/Ch2_In08 *)
    I_111XS2 : BOOL;  (* 111XS2 - Sensor Empurrador Lateral Recuado; at IOBus://rack#0/slot#2/Ch2_In/Ch2_In09 *)
    I_121YS1 : BOOL;  (* 121YS1 - Fotocelula Produto Posicionado BPS1; at IOBus://rack#0/slot#2/Ch2_In/Ch2_In10 *)
    I_121XS1 : BOOL;  (* 121XS1 - Sensor Empurrador Avancado; at IOBus://rack#0/slot#2/Ch2_In/Ch2_In11 *)
    I_121XS2 : BOOL;  (* 121XS2 - Sensor Empurrador Recuado; at IOBus://rack#0/slot#2/Ch2_In/Ch2_In12 *)
    I_122YS1 : BOOL;  (* 122YS1 - Fotocelula Produto Posicionado BPS2; at IOBus://rack#0/slot#2/Ch2_In/Ch2_In13 *)
    I_122XS1 : BOOL;  (* 122XS1 - Sensor Empurrador Avancado; at IOBus://rack#0/slot#2/Ch2_In/Ch2_In14 *)
    I_122XS2 : BOOL;  (* 122XS2 - Sensor Empurrador Recuado; at IOBus://rack#0/slot#2/Ch2_In/Ch2_In15 *)
    I_123YS1 : BOOL;  (* 123YS1 - Fotocelula Produto Posicionado BPS3; at IOBus://rack#0/slot#2/Ch3_In/Ch3_In00 *)
    I_123XS1 : BOOL;  (* 123XS1 - Sensor Empurrador Avancado; at IOBus://rack#0/slot#2/Ch3_In/Ch3_In01 *)
    I_123XS2 : BOOL;  (* 123XS2 - Sensor Empurrador Recuado; at IOBus://rack#0/slot#2/Ch3_In/Ch3_In02 *)
    I_124YS1 : BOOL;  (* 124YS1 - Fotocelula Zona Rejeicao Cheia; at IOBus://rack#0/slot#2/Ch3_In/Ch3_In03 *)
    I_211YS1 : BOOL;  (* 211YS1 - Fotocelula Entrada Transportador; at IOBus://rack#0/slot#2/Ch3_In/Ch3_In04 *)
    I_212YS1 : BOOL;  (* 212YS1 - Fotocelula Entrada Transportador; at IOBus://rack#0/slot#2/Ch3_In/Ch3_In05 *)
    I_213YS1 : BOOL;  (* 213YS1 - Fotocelula Entrada Transportador; at IOBus://rack#0/slot#2/Ch3_In/Ch3_In06 *)
    I_900PS1 : BOOL;  (* 900PS1 - Pressostato Geral de Ar; at IOBus://rack#0/slot#2/Ch3_In/Ch3_In07 *)
    I_211YS2 : BOOL;  (* 211YS2 - Emissor/Recetor Saida Transportador; at IOBus://rack#0/slot#2/Ch4_In/Ch4_In00 *)
    I_211XS1 : BOOL;  (* 211XS1 - Sensor Batente Saida em Cima; at IOBus://rack#0/slot#2/Ch4_In/Ch4_In01 *)
    I_211XS2 : BOOL;  (* 211XS2 - Sensor Batente Saida em Baixo; at IOBus://rack#0/slot#2/Ch4_In/Ch4_In02 *)
    I_212YS2 : BOOL;  (* 212YS2 - Emissor/Recetor Saida Transportador; at IOBus://rack#0/slot#2/Ch4_In/Ch4_In03 *)
    I_212XS1 : BOOL;  (* 212XS1 - Sensor Batente Saida em Cima; at IOBus://rack#0/slot#2/Ch4_In/Ch4_In04 *)
    I_212XS2 : BOOL;  (* 212XS2 - Sensor Batente Saida em Baixo; at IOBus://rack#0/slot#2/Ch4_In/Ch4_In05 *)
    I_213YS2 : BOOL;  (* 213YS2 - Emissor/Recetor Saida Transportador; at IOBus://rack#0/slot#2/Ch4_In/Ch4_In06 *)
    I_213XS1 : BOOL;  (* 213XS1 - Sensor Batente Saida em Cima; at IOBus://rack#0/slot#2/Ch4_In/Ch4_In07 *)
    I_213XS2 : BOOL;  (* 213XS2 - Sensor Batente Saida em Baixo; at IOBus://rack#0/slot#2/Ch4_In/Ch4_In08 *)
    I_221YS2 : BOOL;  (* 221YS2 - Fotocelula Saida Transportador; at IOBus://rack#0/slot#2/Ch4_In/Ch4_In09 *)
    I_222YS2 : BOOL;  (* 222YS2 - Fotocelula Saida Transportador; at IOBus://rack#0/slot#2/Ch4_In/Ch4_In10 *)
    I_223YS3 : BOOL;  (* 223YS3 - Fotocelula Saida Transportador; at IOBus://rack#0/slot#2/Ch4_In/Ch4_In11 *)
    I_230YS2 : BOOL;  (* 230YS2 - Fotocelula Saida Transportador; at IOBus://rack#0/slot#2/Ch4_In/Ch4_In12 *)
    I_231YS1 : BOOL;  (* 231YS1 - Fotocelula Zona Rejeicao Cheia; at IOBus://rack#0/slot#2/Ch4_In/Ch4_In13 *)
    I_240YS2 : BOOL;  (* 240YS2 - Fotocelula Saida Transportador; at IOBus://rack#0/slot#2/Ch4_In/Ch4_In14 *)
    I_250U1OK : BOOL;  (* 250U1OK - Output Leitura OK (Output 1); at IOBus://rack#0/slot#2/Ch4_In/Ch4_In15 *)
    I_250YS1 : BOOL;  (* 250YS1 - Fotocelula Posição Leitura Codigo Barras; at IOBus://rack#0/slot#3/Ch1_In/Ch1_In01 *)
    I_250YS2 : BOOL;  (* 250YS2 - Fotocelula Produto Posicionado; at IOBus://rack#0/slot#3/Ch1_In/Ch1_In02 *)
    I_251XS1 : BOOL;  (* 251XS1 - Sensor Indexador Frontal Avancado; at IOBus://rack#0/slot#3/Ch1_In/Ch1_In03 *)
    I_251XS2 : BOOL;  (* 251XS2 - Sensor Indexador Frontal Recuado; at IOBus://rack#0/slot#3/Ch1_In/Ch1_In04 *)
    I_251YS1 : BOOL;  (* 251YS1 - Fotocelula Produto Posicionado; at IOBus://rack#0/slot#3/Ch1_In/Ch1_In05 *)
    I_252XS1 : BOOL;  (* 252XS1 - Sensor Indexador Lateral Avancado; at IOBus://rack#0/slot#3/Ch1_In/Ch1_In06 *)
    I_252XS2 : BOOL;  (* 252XS2 - Sensor Indexador Lateral Recuado; at IOBus://rack#0/slot#3/Ch1_In/Ch1_In07 *)
    I_310YS2 : BOOL;  (* 310YS2 - Fotocelula Espelho Saida Produto; at IOBus://rack#0/slot#3/Ch2_In/Ch2_In00 *)
    I_320XS1 : BOOL;  (* 320XS1 - Indutivo Posicao Servo Limite Negativo; at IOBus://rack#0/slot#3/Ch2_In/Ch2_In02 *)
    I_320XS2 : BOOL;  (* 320XS2 - Indutivo Posicao Servo Home; at IOBus://rack#0/slot#3/Ch2_In/Ch2_In03 *)
    I_320XS3 : BOOL;  (* 320XS3 - Indutivo Posicao Servo Limite Positivo; at IOBus://rack#0/slot#3/Ch2_In/Ch2_In04 *)
    I_321XS1 : BOOL;  (* 321XS1 - Sensor Inclinador Transportador em Cima; at IOBus://rack#0/slot#3/Ch2_In/Ch2_In05 *)
    I_321XS2 : BOOL;  (* 321XS2 - Sensor Inclinador Transportador em Baixo; at IOBus://rack#0/slot#3/Ch2_In/Ch2_In06 *)
    I_400Auto : BOOL;  (* 400Auto - Ulma em Automatico (Ready to Receive); at IOBus://rack#0/slot#3/Ch2_In/Ch2_In07 *)
    I_530YS1 : BOOL;  (* 530YS1 - Fotocelula Posição Leitura Codigo Barras; at IOBus://rack#0/slot#3/Ch3_In/Ch3_In00 *)
    I_530YS2 : BOOL;  (* 530YS2 - Posição Impressora/Etiquetadora; at IOBus://rack#0/slot#3/Ch3_In/Ch3_In01 *)
    I_530YS3 : BOOL;  (* 530YS3 - Fotocelula Saida Transportador; at IOBus://rack#0/slot#3/Ch3_In/Ch3_In02 *)
    I_530U1OK : BOOL;  (* 530U1OK - Output Leitura OK (Output 1); at IOBus://rack#0/slot#3/Ch3_In/Ch3_In03 *)
    I_530U2OK : BOOL;  (* 530U2OK - Output Leitura OK (Output 1); at IOBus://rack#0/slot#3/Ch3_In/Ch3_In05 *)
    I_550YS1 : BOOL;  (* 550YS1 - Fotocelula Fim de Rolo; at IOBus://rack#0/slot#3/Ch3_In/Ch3_In07 *)
    I_550Feed : BOOL;  (* 550Feed - Sinal Impressora Feed; at IOBus://rack#0/slot#3/Ch3_In/Ch3_In08 *)
    I_550Error : BOOL;  (* 550Error - Sinal Impressora Erro; at IOBus://rack#0/slot#3/Ch3_In/Ch3_In09 *)
    MachineAuto : BOOL;  (* Máquina em automatico; published *)
    MachineOn : BOOL;  (* Máquina Ligada; published *)
    Zona110Auto : BOOL;  (* Zona em Automatico; published *)
    DT_110M1 : DataTransport;
END_VAR
VAR_GLOBAL RETAIN
    G_110V : GrafcetBatente;
END_VAR
VAR_GLOBAL
    Zona120Auto : BOOL;  (* Zona em Automatico; published *)
    Exec_G_110V : BOOL;  (* Executa Grafcet *)
    I_553XS2 : BOOL;  (* 553XS2 - Sensor Empurrador Etiquetas Recuado; at IOBus://rack#0/slot#3/Ch3_In/Ch3_In12 *)
    CondGeraisOK : BOOL;  (* Condições Gerais OK para funcionamento; published *)
    I_650YS1 : BOOL;  (* 650YS1 - Fotocelula Zona Rejeicao Cheia; at IOBus://rack#0/slot#3/Ch3_In/Ch3_In13 *)
    Q_110V1 : BOOL;  (* 110V1 - Valvula Batente Saida Transportador Subir; at IOBus://rack#0/slot#4/Ch1_Out/Ch1_Out00 *)
    Q_110V2 : BOOL;  (* 110V2 - Valvula Batente Saida Transportador Descer; at IOBus://rack#0/slot#4/Ch1_Out/Ch1_Out01 *)
    Q_111U1TRG : BOOL;  (* 111U1TRG - Leitor Código Barras Trigger; at IOBus://rack#0/slot#4/Ch1_Out/Ch1_Out02 *)
    Q_111V1 : BOOL;  (* 111V1 - Valvula Empurrador Lateral Avancado; at IOBus://rack#0/slot#4/Ch1_Out/Ch1_Out03 *)
    Q_111V2 : BOOL;  (* 111V2 - Valvula Empurrador Lateral Recuado; at IOBus://rack#0/slot#4/Ch1_Out/Ch1_Out04 *)
    Q_121V1 : BOOL;  (* 121V1 - Valvula Empurrador Lateral Avancado; at IOBus://rack#0/slot#4/Ch1_Out/Ch1_Out05 *)
    Q_121V2 : BOOL;  (* 121V2 - Valvula Empurrador Lateral Recuado; at IOBus://rack#0/slot#4/Ch1_Out/Ch1_Out06 *)
    Q_122V1 : BOOL;  (* 122V1 - Valvula Empurrador Lateral Avancado; at IOBus://rack#0/slot#4/Ch1_Out/Ch1_Out07 *)
    Q_122V2 : BOOL;  (* 122V2 - Valvula Empurrador Lateral Recuado; at IOBus://rack#0/slot#4/Ch1_Out/Ch1_Out08 *)
    Q_123V1 : BOOL;  (* 123V1 - Valvula Empurrador Lateral Avancado; at IOBus://rack#0/slot#4/Ch1_Out/Ch1_Out09 *)
    Q_123V2 : BOOL;  (* 123V2 - Valvula Empurrador Lateral Recuado; at IOBus://rack#0/slot#4/Ch1_Out/Ch1_Out10 *)
    Q_900V1 : BOOL;  (* 900V1 - Valvula Geral Ar Comprimido; at IOBus://rack#0/slot#4/Ch1_Out/Ch1_Out11 *)
    Q_211V1 : BOOL;  (* 211V1 - Valvula Batente Saida Transportador Subir; at IOBus://rack#0/slot#4/Ch2_Out/Ch2_Out00 *)
    Q_211V2 : BOOL;  (* 211V2 - Valvula Batente Saida Transportador Descer; at IOBus://rack#0/slot#4/Ch2_Out/Ch2_Out01 *)
    Q_212V1 : BOOL;  (* 212V1 - Valvula Batente Saida Transportador Subir; at IOBus://rack#0/slot#4/Ch2_Out/Ch2_Out02 *)
    Q_212V2 : BOOL;  (* 212V2 - Valvula Batente Saida Transportador Descer; at IOBus://rack#0/slot#4/Ch2_Out/Ch2_Out03 *)
    Q_213V1 : BOOL;  (* 213V1 - Valvula Batente Saida Transportador Subir; at IOBus://rack#0/slot#4/Ch2_Out/Ch2_Out04 *)
    Q_213V2 : BOOL;  (* 213V2 - Valvula Batente Saida Transportador Descer; at IOBus://rack#0/slot#4/Ch2_Out/Ch2_Out05 *)
    Q_250U1TRG : BOOL;  (* 250U1TRG - Leitor Código Barras Trigger; at IOBus://rack#0/slot#4/Ch2_Out/Ch2_Out06 *)
    Q_251V1 : BOOL;  (* 251V1 - Valvula Indexador Lateral Avancado; at IOBus://rack#0/slot#4/Ch2_Out/Ch2_Out07 *)
    Q_251V2 : BOOL;  (* 251V2 - Valvula Indexador Lateral Recuado; at IOBus://rack#0/slot#4/Ch2_Out/Ch2_Out08 *)
    Q_252V1 : BOOL;  (* 252V1 - Valvula Indexador Frontal Avancado; at IOBus://rack#0/slot#4/Ch2_Out/Ch2_Out09 *)
    Q_252V2 : BOOL;  (* 252V2 - Valvula Indexador Frontal Recuado; at IOBus://rack#0/slot#4/Ch2_Out/Ch2_Out10 *)
    Q_310VL1 : BOOL;  (* 310VL1 - Smart Motor Velocidade 1; at IOBus://rack#0/slot#4/Ch3_Out/Ch3_Out00 *)
    Q_310VL2 : BOOL;  (* 310VL2 - Smart Motor Velocidade 2; at IOBus://rack#0/slot#4/Ch3_Out/Ch3_Out01 *)
    Q_320XS1 : BOOL;  (* 320XS1 - Posicao Servo Limite Negativo; at IOBus://rack#0/slot#4/Ch3_Out/Ch3_Out02 *)
    Q_320XS2 : BOOL;  (* 320XS2 - Posicao Servo Home; at IOBus://rack#0/slot#4/Ch3_Out/Ch3_Out03 *)
    Q_320XS3 : BOOL;  (* 320XS3 - Posicao Servo Limite Positivo; at IOBus://rack#0/slot#4/Ch3_Out/Ch3_Out04 *)
    Q_321V1 : BOOL;  (* 321V1 - Valvula Inclinador Transportador Subir; at IOBus://rack#0/slot#4/Ch3_Out/Ch3_Out05 *)
    Q_321V2 : BOOL;  (* 321V2 - Valvula Inclinador Transportador Descer; at IOBus://rack#0/slot#4/Ch3_Out/Ch3_Out06 *)
    Q_900LG : BOOL;  (* 900LG - Sinalizacao Verde; at IOBus://rack#0/slot#4/Ch3_Out/Ch3_Out10 *)
    Q_900LR : BOOL;  (* 900LR - Sinalizacao Vermelho; at IOBus://rack#0/slot#4/Ch3_Out/Ch3_Out11 *)
    Q_520V1 : BOOL;  (* 520V1 - Valvula Transferencia Subir; at IOBus://rack#0/slot#4/Ch4_Out/Ch4_Out00 *)
    Q_520V2 : BOOL;  (* 520V2 - Valvula Transferencia Descer; at IOBus://rack#0/slot#4/Ch4_Out/Ch4_Out01 *)
    Q_530VL1 : BOOL;  (* 530VL1 - Smart Motor Velocidade 1; at IOBus://rack#0/slot#4/Ch4_Out/Ch4_Out02 *)
    Q_530VL2 : BOOL;  (* 530VL2 - Smart Motor Velocidade 2; at IOBus://rack#0/slot#4/Ch4_Out/Ch4_Out03 *)
    Q_530U1TRG : BOOL;  (* 530U1TRG - Leitor Código Barras Trigger; at IOBus://rack#0/slot#4/Ch4_Out/Ch4_Out04 *)
    Q_530U2TRG : BOOL;  (* 530U2TRG - Leitor Código Barras Trigger; at IOBus://rack#0/slot#4/Ch4_Out/Ch4_Out05 *)
    Q_540V1 : BOOL;  (* 540V1 - Valvula Transferencia Subir; at IOBus://rack#0/slot#4/Ch4_Out/Ch4_Out06 *)
    Q_540V2 : BOOL;  (* 540V2 - Valvula Transferencia Descer; at IOBus://rack#0/slot#4/Ch4_Out/Ch4_Out07 *)
    Q_550M1 : BOOL;  (* 550M1 - Motor Rebobinador; at IOBus://rack#0/slot#4/Ch4_Out/Ch4_Out08 *)
    Q_550LG : BOOL;  (* 550LG - Sinalizacao Verde; at IOBus://rack#0/slot#4/Ch4_Out/Ch4_Out09 *)
    Q_550LR : BOOL;  (* 550LR - Sinalizacao Vermelho; at IOBus://rack#0/slot#4/Ch4_Out/Ch4_Out10 *)
    Q_551V1 : BOOL;  (* 551V1 - Valvula Venturi Vacuo; at IOBus://rack#0/slot#4/Ch4_Out/Ch4_Out11 *)
    Q_552V1 : BOOL;  (* 552V1 - Valvula Sopro Etiqueta; at IOBus://rack#0/slot#4/Ch4_Out/Ch4_Out12 *)
    Q_553V1 : BOOL;  (* 553V1 - Valvula Empurrador Etiqueta Avancado; at IOBus://rack#0/slot#4/Ch4_Out/Ch4_Out13 *)
    Q_553V2 : BOOL;  (* 553V2 - Valvula Empurrador Etiqueta Recuado; at IOBus://rack#0/slot#4/Ch4_Out/Ch4_Out14 *)
    Q_641V1 : BOOL;  (* 641V1 - Valvula Transferencia Subir; at IOBus://rack#0/slot#4/Ch4_Out/Ch4_Out15 *)
    Q_641V2 : BOOL;  (* 641V2 - Valvula Transferencia Descer; at IOBus://rack#0/slot#5/Ch1_Out/Ch1_Out00 *)
    Q_642V1 : BOOL;  (* 642V1 - Valvula Transferencia Subir; at IOBus://rack#0/slot#5/Ch1_Out/Ch1_Out01 *)
    Q_642V2 : BOOL;  (* 642V2 - Valvula Transferencia Descer; at IOBus://rack#0/slot#5/Ch1_Out/Ch1_Out02 *)
    Q_643V1 : BOOL;  (* 643V1 - Valvula Transferencia Subir; at IOBus://rack#0/slot#5/Ch1_Out/Ch1_Out03 *)
    Q_643V2 : BOOL;  (* 643V2 - Valvula Transferencia Descer; at IOBus://rack#0/slot#5/Ch1_Out/Ch1_Out04 *)
    IFQ_330_NotaType AT %404 : WORD;  (* Tipo de Nota para Robot *)
    IFI_330_NotaType AT %204 : WORD;  (* Tipo de Nota do Robot; published *)
    IFI_330_WatchDog : BOOL;  (* 330 - WatchDog; published *)
    IFI_330_In310 : BOOL;  (* 330 - Robot na Zona 310; published *)
    IFI_330_In250 : BOOL;  (* 330 - Robot na Zona 250; published *)
    E002_RPDO4_mapping_parameter_CiA_Controlword_6040_00 : UINT;  (* at ECAT://node#11/RPDO4 mapping parameter_CiA: Controlword_6040_00 *)
    E002_RPDO4_mapping_parameter_Target_velocity_6042_00 : INT;  (* at ECAT://node#11/RPDO4 mapping parameter_Target velocity_6042_00 *)
    D_110M1 : DataMotor;  (* Data Motor; published *)
    D_111M1 : DataMotor;  (* Data Motor; published *)
    A_110M1 : AlarmeGeralEquipamento;  (* published *)
    A_111M1 : AlarmeGeralEquipamento;  (* published *)
    E_110M1 : Event;  (* Event; published *)
    E_111M1 : Event;  (* Event; published *)
    E002_TPDO4_mapping_parameter_CiA_Statusword_6041_00 : UINT;  (* at ECAT://node#11/TPDO4 mapping parameter_CiA: Statusword_6041_00 *)
    E003_RPDO4_mapping_parameter_CiA_Controlword_6040_00 : UINT;  (* at ECAT://node#12/RPDO4 mapping parameter_CiA: Controlword_6040_00 *)
    E003_RPDO4_mapping_parameter_Target_velocity_6042_00 : INT;  (* at ECAT://node#12/RPDO4 mapping parameter_Target velocity_6042_00 *)
    E003_TPDO4_mapping_parameter_CiA_Statusword_6041_00 : UINT;  (* at ECAT://node#12/TPDO4 mapping parameter_CiA: Statusword_6041_00 *)
    E004_RPDO4_mapping_parameter_CiA_Controlword_6040_00 : UINT;  (* at ECAT://node#13/RPDO4 mapping parameter_CiA: Controlword_6040_00 *)
    E004_RPDO4_mapping_parameter_Target_velocity_6042_00 : INT;  (* at ECAT://node#13/RPDO4 mapping parameter_Target velocity_6042_00 *)
    E004_TPDO4_mapping_parameter_CiA_Statusword_6041_00 : UINT;  (* at ECAT://node#13/TPDO4 mapping parameter_CiA: Statusword_6041_00 *)
    E005_RPDO4_mapping_parameter_CiA_Controlword_6040_00 : UINT;  (* at ECAT://node#14/RPDO4 mapping parameter_CiA: Controlword_6040_00 *)
    E005_RPDO4_mapping_parameter_Target_velocity_6042_00 : INT;  (* at ECAT://node#14/RPDO4 mapping parameter_Target velocity_6042_00 *)
    E005_TPDO4_mapping_parameter_CiA_Statusword_6041_00 : UINT;  (* at ECAT://node#14/TPDO4 mapping parameter_CiA: Statusword_6041_00 *)
    E006_RPDO4_mapping_parameter_CiA_Controlword_6040_00 : UINT;  (* at ECAT://node#15/RPDO4 mapping parameter_CiA: Controlword_6040_00 *)
    E006_RPDO4_mapping_parameter_Target_velocity_6042_00 : INT;  (* at ECAT://node#15/RPDO4 mapping parameter_Target velocity_6042_00 *)
    E006_TPDO4_mapping_parameter_CiA_Statusword_6041_00 : UINT;  (* at ECAT://node#15/TPDO4 mapping parameter_CiA: Statusword_6041_00 *)
    E007_RPDO4_mapping_parameter_CiA_Controlword_6040_00 : UINT;  (* at ECAT://node#16/RPDO4 mapping parameter_CiA: Controlword_6040_00 *)
    E007_RPDO4_mapping_parameter_Target_velocity_6042_00 : INT;  (* at ECAT://node#16/RPDO4 mapping parameter_Target velocity_6042_00 *)
    E007_TPDO4_mapping_parameter_CiA_Statusword_6041_00 : UINT;  (* at ECAT://node#16/TPDO4 mapping parameter_CiA: Statusword_6041_00 *)
    E008_RPDO4_mapping_parameter_CiA_Controlword_6040_00 : UINT;  (* at ECAT://node#21/RPDO4 mapping parameter_CiA: Controlword_6040_00 *)
    E008_RPDO4_mapping_parameter_Target_velocity_6042_00 : INT;  (* at ECAT://node#21/RPDO4 mapping parameter_Target velocity_6042_00 *)
    E008_TPDO4_mapping_parameter_CiA_Statusword_6041_00 : UINT;  (* at ECAT://node#21/TPDO4 mapping parameter_CiA: Statusword_6041_00 *)
    E009_RPDO4_mapping_parameter_CiA_Controlword_6040_00 : UINT;  (* at ECAT://node#22/RPDO4 mapping parameter_CiA: Controlword_6040_00 *)
    E009_RPDO4_mapping_parameter_Target_velocity_6042_00 : INT;  (* at ECAT://node#22/RPDO4 mapping parameter_Target velocity_6042_00 *)
    E009_TPDO4_mapping_parameter_CiA_Statusword_6041_00 : UINT;  (* at ECAT://node#22/TPDO4 mapping parameter_CiA: Statusword_6041_00 *)
    E010_RPDO4_mapping_parameter_CiA_Controlword_6040_00 : UINT;  (* at ECAT://node#23/RPDO4 mapping parameter_CiA: Controlword_6040_00 *)
    E010_RPDO4_mapping_parameter_Target_velocity_6042_00 : INT;  (* at ECAT://node#23/RPDO4 mapping parameter_Target velocity_6042_00 *)
    E010_TPDO4_mapping_parameter_CiA_Statusword_6041_00 : UINT;  (* at ECAT://node#23/TPDO4 mapping parameter_CiA: Statusword_6041_00 *)
    E011_RPDO4_mapping_parameter_CiA_Controlword_6040_00 : UINT;  (* at ECAT://node#24/RPDO4 mapping parameter_CiA: Controlword_6040_00 *)
    E011_RPDO4_mapping_parameter_Target_velocity_6042_00 : INT;  (* at ECAT://node#24/RPDO4 mapping parameter_Target velocity_6042_00 *)
    E011_TPDO4_mapping_parameter_CiA_Statusword_6041_00 : UINT;  (* at ECAT://node#24/TPDO4 mapping parameter_CiA: Statusword_6041_00 *)
    E012_RPDO4_mapping_parameter_CiA_Controlword_6040_00 : UINT;  (* at ECAT://node#25/RPDO4 mapping parameter_CiA: Controlword_6040_00 *)
    E012_RPDO4_mapping_parameter_Target_velocity_6042_00 : INT;  (* at ECAT://node#25/RPDO4 mapping parameter_Target velocity_6042_00 *)
    E012_TPDO4_mapping_parameter_CiA_Statusword_6041_00 : UINT;  (* at ECAT://node#25/TPDO4 mapping parameter_CiA: Statusword_6041_00 *)
    E013_RPDO4_mapping_parameter_CiA_Controlword_6040_00 : UINT;  (* at ECAT://node#26/RPDO4 mapping parameter_CiA: Controlword_6040_00 *)
    E013_RPDO4_mapping_parameter_Target_velocity_6042_00 : INT;  (* at ECAT://node#26/RPDO4 mapping parameter_Target velocity_6042_00 *)
    E013_TPDO4_mapping_parameter_CiA_Statusword_6041_00 : UINT;  (* at ECAT://node#26/TPDO4 mapping parameter_CiA: Statusword_6041_00 *)
    E003_RPDO6_mapping_parameter_CiA_Acceleration_ms_2917_00 : UINT;  (* at ECAT://node#12/RPDO6 mapping parameter_CiA: Acceleration ms_2917_00 *)
    E003_RPDO6_mapping_parameter_CiA_Deceleration_ms_2918_00 : UINT;  (* at ECAT://node#12/RPDO6 mapping parameter_CiA: Deceleration ms_2918_00 *)
    E002_RPDO6_mapping_parameter_CiA_Acceleration_ms_2917_00 : UINT;  (* at ECAT://node#11/RPDO6 mapping parameter_CiA: Acceleration ms_2917_00 *)
    E002_RPDO6_mapping_parameter_CiA_Deceleration_ms_2918_00 : UINT;  (* at ECAT://node#11/RPDO6 mapping parameter_CiA: Deceleration ms_2918_00 *)
    E004_RPDO6_mapping_parameter_CiA_Acceleration_ms_2917_00 : UINT;  (* at ECAT://node#13/RPDO6 mapping parameter_CiA: Acceleration ms_2917_00 *)
    E004_RPDO6_mapping_parameter_CiA_Deceleration_ms_2918_00 : UINT;  (* at ECAT://node#13/RPDO6 mapping parameter_CiA: Deceleration ms_2918_00 *)
    E005_RPDO6_mapping_parameter_CiA_Acceleration_ms_2917_00 : UINT;  (* at ECAT://node#14/RPDO6 mapping parameter_CiA: Acceleration ms_2917_00 *)
    E005_RPDO6_mapping_parameter_CiA_Deceleration_ms_2918_00 : UINT;  (* at ECAT://node#14/RPDO6 mapping parameter_CiA: Deceleration ms_2918_00 *)
    E006_RPDO6_mapping_parameter_CiA_Acceleration_ms_2917_00 : UINT;  (* at ECAT://node#15/RPDO6 mapping parameter_CiA: Acceleration ms_2917_00 *)
    E006_RPDO6_mapping_parameter_CiA_Deceleration_ms_2918_00 : UINT;  (* at ECAT://node#15/RPDO6 mapping parameter_CiA: Deceleration ms_2918_00 *)
    E007_RPDO6_mapping_parameter_CiA_Acceleration_ms_2917_00 : UINT;  (* at ECAT://node#16/RPDO6 mapping parameter_CiA: Acceleration ms_2917_00 *)
    E007_RPDO6_mapping_parameter_CiA_Deceleration_ms_2918_00 : UINT;  (* at ECAT://node#16/RPDO6 mapping parameter_CiA: Deceleration ms_2918_00 *)
    E008_RPDO6_mapping_parameter_CiA_Acceleration_ms_2917_00 : UINT;  (* at ECAT://node#21/RPDO6 mapping parameter_CiA: Acceleration ms_2917_00 *)
    E008_RPDO6_mapping_parameter_CiA_Deceleration_ms_2918_00 : UINT;  (* at ECAT://node#21/RPDO6 mapping parameter_CiA: Deceleration ms_2918_00 *)
    E009_RPDO6_mapping_parameter_CiA_Acceleration_ms_2917_00 : UINT;  (* at ECAT://node#22/RPDO6 mapping parameter_CiA: Acceleration ms_2917_00 *)
    E009_RPDO6_mapping_parameter_CiA_Deceleration_ms_2918_00 : UINT;  (* at ECAT://node#22/RPDO6 mapping parameter_CiA: Deceleration ms_2918_00 *)
    E010_RPDO6_mapping_parameter_CiA_Acceleration_ms_2917_00 : UINT;  (* at ECAT://node#23/RPDO6 mapping parameter_CiA: Acceleration ms_2917_00 *)
    E010_RPDO6_mapping_parameter_CiA_Deceleration_ms_2918_00 : UINT;  (* at ECAT://node#23/RPDO6 mapping parameter_CiA: Deceleration ms_2918_00 *)
    E011_RPDO6_mapping_parameter_CiA_Acceleration_ms_2917_00 : UINT;  (* at ECAT://node#24/RPDO6 mapping parameter_CiA: Acceleration ms_2917_00 *)
    E011_RPDO6_mapping_parameter_CiA_Deceleration_ms_2918_00 : UINT;  (* at ECAT://node#24/RPDO6 mapping parameter_CiA: Deceleration ms_2918_00 *)
    E012_RPDO6_mapping_parameter_CiA_Acceleration_ms_2917_00 : UINT;  (* at ECAT://node#25/RPDO6 mapping parameter_CiA: Acceleration ms_2917_00 *)
    E012_RPDO6_mapping_parameter_CiA_Deceleration_ms_2918_00 : UINT;  (* at ECAT://node#25/RPDO6 mapping parameter_CiA: Deceleration ms_2918_00 *)
    E013_RPDO6_mapping_parameter_CiA_Acceleration_ms_2917_00 : UINT;  (* at ECAT://node#26/RPDO6 mapping parameter_CiA: Acceleration ms_2917_00 *)
    E013_RPDO6_mapping_parameter_CiA_Deceleration_ms_2918_00 : UINT;  (* at ECAT://node#26/RPDO6 mapping parameter_CiA: Deceleration ms_2918_00 *)
    ResetAlarmes : BOOL := False;  (* Reset Alarmes; published *)
    IFQ_330_StopRequest : BOOL;  (* 330 - Pedido de Acesso; published *)
    IFI_330_InHome : BOOL;  (* 330 - Robot em Home Position; published *)
    IFI_330_RstDone : BOOL;  (* 330 - Robot Efetuou Reset ao Ciclo - Espera primeiro milheiro; published *)
    IFI_330_StopRequestDone : BOOL;  (* 330 - Robot Permite Acesso à Zona; published *)
    IFI_330_ProductLost : BOOL;  (* 330 - Robot Perdeu Milheiro ou não está bem posicionado; published *)
    IFI_330_GeneralError : BOOL;  (* 330 - Robot em Erro Geral - Verificar Consola do Robot; published *)
    IFI_330_BoxComplete : BOOL;  (* 330 - Robot Finalizou Entrega 10 Milheiros; published *)
    IFI_330_OpenTool : BOOL;  (* 330 - Robot Pede Abertura Ferramenta; published *)
    IFI_330_CloseTool : BOOL;  (* 330 - Robot Pede Fecho Ferramenta; published *)
    IFQ_330_330YS1 : BOOL;  (* 330 - Imagem de 310YS1; published *)
    IFQ_330_330YS2 : BOOL;  (* 330 - Imagem de 310YS2; published *)
    IFQ_330_330XS1 : BOOL;  (* 330 - Imagem de 310XS1; published *)
    IFQ_330_RstProdLost : BOOL;  (* 330 - Reset Erro Perda de Milheiro; published *)
    Q_330V2 : BOOL;  (* 330V2 - Valvula Ferramenta Robot Fechar; at IOBus://rack#0/slot#4/Ch3_Out/Ch3_Out13 *)
    I_330YS1 : BOOL;  (* 330YS1 - Fotocelula Presença Produto; at IOBus://rack#0/slot#3/Ch2_In/Ch2_In08 *)
    I_330YS2 : BOOL;  (* 330YS2 - Fotocelula Presença Produto; at IOBus://rack#0/slot#3/Ch2_In/Ch2_In09 *)
    I_330XS1 : BOOL;  (* 330XS1 - Sensor Ferramenta Robot Aberto; at IOBus://rack#0/slot#3/Ch2_In/Ch2_In10 *)
    A_120M1 : AlarmeGeralEquipamento;  (* published *)
    A_211M1 : AlarmeGeralEquipamento;  (* published *)
    A_212M1 : AlarmeGeralEquipamento;  (* published *)
    A_213M1 : AlarmeGeralEquipamento;  (* published *)
    A_221M1 : AlarmeGeralEquipamento;  (* published *)
    A_222M1 : AlarmeGeralEquipamento;  (* published *)
    A_223M1 : AlarmeGeralEquipamento;  (* published *)
    A_230M1 : AlarmeGeralEquipamento;  (* published *)
    A_240M1 : AlarmeGeralEquipamento;  (* published *)
    A_250M1 : AlarmeGeralEquipamento;  (* published *)
    A_310M1 : AlarmeGeralEquipamento;  (* published *)
    A_510M1 : AlarmeGeralEquipamento;  (* published *)
    A_520M1 : AlarmeGeralEquipamento;  (* published *)
    A_520M2 : AlarmeGeralEquipamento;  (* published *)
    A_530M1 : AlarmeGeralEquipamento;  (* published *)
    A_540M1 : AlarmeGeralEquipamento;  (* published *)
    A_540M2 : AlarmeGeralEquipamento;  (* published *)
    A_610M1 : AlarmeGeralEquipamento;  (* published *)
    A_620M1 : AlarmeGeralEquipamento;  (* published *)
    A_630M1 : AlarmeGeralEquipamento;  (* published *)
    A_640M1 : AlarmeGeralEquipamento;  (* published *)
    A_640M2 : AlarmeGeralEquipamento;  (* published *)
    A_641M1 : AlarmeGeralEquipamento;  (* published *)
    A_642M1 : AlarmeGeralEquipamento;  (* published *)
    A_643M1 : AlarmeGeralEquipamento;  (* published *)
    D_120M1 : DataMotor;  (* Data Motor; published *)
    D_211M1 : DataMotor;  (* Data Motor; published *)
    D_212M1 : DataMotor;  (* Data Motor; published *)
    D_213M1 : DataMotor;  (* Data Motor; published *)
    D_221M1 : DataMotor;  (* Data Motor; published *)
    D_222M1 : DataMotor;  (* Data Motor; published *)
    D_223M1 : DataMotor;  (* Data Motor; published *)
    D_230M1 : DataMotor;  (* Data Motor; published *)
    D_240M1 : DataMotor;  (* Data Motor; published *)
    D_250M1 : DataMotor;  (* Data Motor; published *)
    D_310M1 : DataMotor;  (* Data Motor; published *)
    D_510M1 : DataMotor;  (* Data Motor; published *)
    D_520M1 : DataMotor;  (* Data Motor; published *)
    D_520M2 : DataMotor;  (* Data Motor; published *)
    D_530M1 : DataMotor;  (* Data Motor; published *)
    D_540M1 : DataMotor;  (* Data Motor; published *)
    D_540M2 : DataMotor;  (* Data Motor; published *)
    D_610M1 : DataMotor;  (* Data Motor; published *)
    D_620M1 : DataMotor;  (* Data Motor; published *)
    D_630M1 : DataMotor;  (* Data Motor; published *)
    D_640M1 : DataMotor;  (* Data Motor; published *)
    D_640M2 : DataMotor;  (* Data Motor; published *)
    D_641M1 : DataMotor;  (* Data Motor; published *)
    D_642M1 : DataMotor;  (* Data Motor; published *)
    D_643M1 : DataMotor;  (* Data Motor; published *)
    E_120M1 : Event;  (* Event; published *)
    E_211M1 : Event;  (* Event; published *)
    E_212M1 : Event;  (* Event; published *)
    E_213M1 : Event;  (* Event; published *)
    E_221M1 : Event;  (* Event; published *)
    E_222M1 : Event;  (* Event; published *)
    E_223M1 : Event;  (* Event; published *)
    E_230M1 : Event;  (* Event; published *)
    E_240M1 : Event;  (* Event; published *)
    E_250M1 : Event;  (* Event; published *)
    E_310M1 : Event;  (* Event; published *)
    E_510M1 : Event;  (* Event; published *)
    E_520M1 : Event;  (* Event; published *)
    E_520M2 : Event;  (* Event; published *)
    E_540M1 : Event;  (* Event; published *)
    E_540M2 : Event;  (* Event; published *)
    E_610M1 : Event;  (* Event; published *)
    E_620M1 : Event;  (* Event; published *)
    E_630M1 : Event;  (* Event; published *)
    E_640M1 : Event;  (* Event; published *)
    E_640M2 : Event;  (* Event; published *)
    E_641M1 : Event;  (* Event; published *)
    E_642M1 : Event;  (* Event; published *)
    E_643M1 : Event;  (* Event; published *)
    T_Reset : BOOL;  (* Sinal de Teste - Comissionamento; at IOBus://rack#0/slot#2/Ch1_In/Ch1_In13 *)
    Exec_G_111V : BOOL;  (* Executa Grafcet *)
    ZonaBuffer1Auto : BOOL;  (* Zona em Automatico; published *)
    ZonaBuffer2Auto : BOOL;  (* Zona em Automatico; published *)
    ZonaBuffer3Auto : BOOL;  (* Zona em Automatico; published *)
    Exec_G_121V : BOOL;  (* Executa Grafcet *)
    Exec_G_122V : BOOL;  (* Executa Grafcet *)
    Exec_G_123V : BOOL;  (* Executa Grafcet *)
END_VAR
VAR_GLOBAL RETAIN
    G_121V : GrafcetEmpurrador;
    G_122V : GrafcetEmpurrador;
    G_123V : GrafcetEmpurrador;
END_VAR
VAR_GLOBAL
    Exec_G_211V : BOOL;  (* Executa Grafcet *)
    Exec_G_212V : BOOL;  (* Executa Grafcet *)
    Exec_G_213V : BOOL;  (* Executa Grafcet *)
END_VAR
VAR_GLOBAL RETAIN
    G_211V : GrafcetBatente;
    G_212V : GrafcetBatente;
    G_213V : GrafcetBatente;
END_VAR
VAR_GLOBAL
    DT_211M1 : DataTransport;
END_VAR
VAR_GLOBAL RETAIN
    DP_221M1 : DataProd;  (* published *)
    DP_222M1 : DataProd;  (* published *)
    DP_223M1 : DataProd;  (* published *)
END_VAR
VAR_GLOBAL
    DT_212M1 : DataTransport;
    DT_213M1 : DataTransport;
    Exec_G_221M1 : BOOL;  (* Executa Grafcet *)
    Exec_G_222M1 : BOOL;  (* Executa Grafcet *)
    Exec_G_223M1 : BOOL;  (* Executa Grafcet *)
END_VAR
VAR_GLOBAL RETAIN
    G_221M1 : GrafcetAcumula;
    G_222M1 : GrafcetAcumula;
    G_223M1 : GrafcetAcumula;
END_VAR
VAR_GLOBAL
    AG_221M1 : Alarme;  (* published *)
END_VAR
VAR_GLOBAL RETAIN
    DP_211M1 : DataProd;  (* published *)
    DP_212M1 : DataProd;  (* published *)
    DP_213M1 : DataProd;  (* published *)
END_VAR
VAR_GLOBAL
    Zona230Auto : BOOL;  (* Zona em Automatico; published *)
    AG_222M1 : Alarme;  (* published *)
    AG_223M1 : Alarme;  (* published *)
    AG_230M1 : Alarme;  (* published *)
    AG_240M1 : Alarme;  (* published *)
    AG_250M1 : Alarme;  (* published *)
END_VAR
VAR_GLOBAL RETAIN
    G_230M1 : Grafcet230M1;
END_VAR
VAR_GLOBAL
    Exec_G_230M1 : BOOL;  (* Executa Grafcet *)
    Exec_G_240M1 : BOOL;  (* Executa Grafcet *)
    Exec_G_250M1 : BOOL;  (* Executa Grafcet *)
END_VAR
VAR_GLOBAL RETAIN
    DP_230M1 : DataProd;  (* published *)
    DP_240M1 : DataProd;  (* published *)
    DP_250M1 : DataProd;  (* published *)
    G_240M1 : Grafcet240M1;
END_VAR
VAR_GLOBAL
    Zona240Auto : BOOL;  (* Zona em Automatico; published *)
    Zona250Auto : BOOL;  (* Zona em Automatico; published *)
END_VAR
VAR_GLOBAL RETAIN
    G_250M1 : Grafcet250M1;
END_VAR
VAR_GLOBAL
    Q_Interroll_540 : Out_EIPMulticontrol;  (* network output *)
    Q_Interroll_520 : Out_EIPMulticontrol;  (* network output *)
    Q_Interroll_641 : Out_EIPMulticontrol;  (* network output *)
    I_Interroll_540 : In_EIPMulticontrol;  (* network input *)
    I_Interroll_641 : In_EIPMulticontrol;  (* network input *)
    Q_Interroll_643 : Out_EIPMulticontrol;  (* network output *)
    I_Interroll_643 : In_EIPMulticontrol;  (* network input *)
    I_Interroll_520 : In_EIPMulticontrol;  (* network input *)
    I_FromG9SP_100 : ARRAY[0..67] OF byte;  (* network input *)
    Q_ToG9SP_101 : ARRAY[0..5] OF byte;  (* network output *)
    I_IFM01_BarCodeReader_250U1 : ARRAY[0..449] OF BYTE;  (* network input *)
    I_IFM01_BarCodeReader_530U1 : ARRAY[0..449] OF BYTE;  (* network input *)
    I_IFM01_BarCodeReader_530U2 : ARRAY[0..449] OF BYTE;  (* network input *)
    I_IFM01_BarCodeReader_111U1 : ARRAY[0..449] OF BYTE;  (* network input *)
    Exec_G_111M1 : BOOL;  (* Executa Grafcet *)
    Exec_G_120M1 : BOOL;  (* Executa Grafcet *)
END_VAR
VAR_GLOBAL RETAIN
    G_111M1 : Grafcet111M1;
    G_120M1 : Grafcet120M1;
END_VAR
VAR_GLOBAL
    WatchDogHMI : BOOL;  (* published *)
    DP_120M1 : DataProd;  (* published *)
    DP_111M1 : DataProd;  (* published *)
    DataRead111U1 : DataLCB;  (* published *)
    Exec_G_251V : BOOL;  (* Executa Grafcet *)
    Exec_G_252V : BOOL;  (* Executa Grafcet *)
END_VAR
VAR_GLOBAL RETAIN
    G_251V : GrafcetEmpurrador;
    G_252V : GrafcetEmpurrador;
END_VAR
VAR_GLOBAL
    HMI_EtiquetaMilheiro_01 : STRING[256];  (* published *)
    HMI_EtiquetaMilheiro_02 : STRING[256];  (* published *)
    HMI_EtiquetaMilheiro_03 : STRING[256];  (* published *)
    HMI_EtiquetaMilheiro_04 : STRING[256];  (* published *)
    HMI_EtiquetaMilheiro_05 : STRING[256];  (* published *)
    HMI_EtiquetaMilheiro_06 : STRING[256];  (* published *)
    HMI_EtiquetaMilheiro_07 : STRING[256];  (* published *)
    HMI_EtiquetaMilheiro_08 : STRING[256];  (* published *)
    HMI_EtiquetaMilheiro_09 : STRING[256];  (* published *)
    HMI_EtiquetaMilheiro_10 : STRING[256];  (* published *)
    HMI_PleaseCreateBox : BOOL;  (* published *)
    HMI_PleasePrintBoxId : BOOL;  (* published *)
    HMI_CreateBoxOK : BOOL;  (* published *)
    HMI_CreateBoxNOK : BOOL;  (* published *)
    HMI_PrintOK : BOOL;  (* published *)
    HMI_PrintNOK : BOOL;  (* published *)
    HMI_Maquina : string[256];  (* published *)
END_VAR
VAR_GLOBAL CONSTANT
    MC_Axis320M1 : _sAXIS_REF;  (* at MC://_MC_AX[0] *)
END_VAR
VAR_GLOBAL
    I_540YS1 : BOOL;
    I_540YS2 : BOOL;
    I_540XS1 : BOOL;
    I_540XS2 : BOOL;
    D_320M1 : DataServo;
    E015_Error_code : WORD;  (* at ECAT://node#31/Error code *)
    Exec_G_310M1 : BOOL;  (* Executa Grafcet *)
    Zona310Auto : BOOL;  (* Zona em Automatico; published *)
END_VAR
VAR_GLOBAL RETAIN
    G_310M1 : Grafcet310M1;
END_VAR
VAR_GLOBAL
    AG_310M1 : Alarme;  (* published *)
END_VAR
VAR_GLOBAL RETAIN
    DP_320M1 : Position;  (* published *)
    WidthMax320M1 : LREAL;  (* Distância do ponto zero ao Batente; published *)
    Width5Euro : LREAL;  (* Largura Nota 5 Euros; published *)
    Width10Euro : LREAL;  (* Largura Nota 10 Euros; published *)
    Width20Euro : LREAL;  (* Largura Nota 20 Euros; published *)
    Width50Euro : LREAL;  (* Largura Nota 50 Euros; published *)
    Width100Euro : LREAL;  (* Largura Nota 100 Euros; published *)
    Width200Euro : LREAL;  (* Largura Nota 200 Euros; published *)
    Width500Euro : LREAL;  (* Largura Nota 500 Euros; published *)
    DP_310M1 : DataProd;
END_VAR
VAR_GLOBAL
    DataRead250U1 : DataLCB;  (* published *)
    DataRead530U1 : DataLCB;  (* published *)
    DataRead530U2 : DataLCB;  (* published *)
    Code111U1OK : BOOL;  (* Código Valido *)
    Code111U1NOK : BOOL;  (* Código Não Valido *)
    Code250U1OK : BOOL;  (* Código Valido *)
    Code250U1NOK : BOOL;  (* Código Não Valido *)
END_VAR
VAR_GLOBAL RETAIN
    G_111U1 : Grafcet111U1;
    G_250U1 : Grafcet250U1;
END_VAR
VAR_GLOBAL
    A_111U1 : Alarme;  (* published *)
    A_250U1 : Alarme;  (* published *)
    Exec_G_111U1 : BOOL;  (* Executa Grafcet *)
    Exec_G_250U1 : BOOL;  (* Executa Grafcet *)
    TRG_111U1 : BOOL;  (* Trigger Leitor Código de Barras *)
    TRG_250U1 : BOOL;  (* Trigger Leitor Código de Barras *)
    Erro_111U1 : BOOL;  (* Erro no código de barras *)
    Erro_250U1 : BOOL;  (* Erro no código de barras *)
    JulianDateES1 : UINT;  (* Data Juliana Notas Serie 1 *)
    JulianDateES2 : UINT;  (* Data Juliana Notas Serie 2 *)
    ds : _sDT;  (* DateStruct of the Var SystemTime to use on "Julian Date" *)
END_VAR
VAR_GLOBAL RETAIN
    D_Buffer1 : DataBuffer;  (* published *)
    D_Buffer2 : DataBuffer;  (* published *)
    D_Buffer3 : DataBuffer;  (* published *)
END_VAR
VAR_GLOBAL
    ErroComunicacaoPC : BOOL;  (* published *)
    Exec_G_510M1 : BOOL;  (* Executa Grafcet *)
END_VAR
VAR_GLOBAL RETAIN
    G_510M1 : Grafcet510M1;
END_VAR
VAR_GLOBAL
    I_510YS2 : BOOL;
    I_510YS1 : BOOL;
END_VAR
VAR_GLOBAL RETAIN
    G_520M1 : Grafcet520M1;
END_VAR
VAR_GLOBAL
    Exec_G_520M1 : BOOL;  (* Executa Grafcet *)
    I_520XS1 : BOOL;
    I_520XS2 : BOOL;
    Zona510520Auto : BOOL;  (* Zona em Automatico; published *)
    I_520YS1 : BOOL;
END_VAR
VAR_GLOBAL RETAIN
    G_530M1 : Grafcet530M1;
END_VAR
VAR_GLOBAL
    Exec_G_530M1 : BOOL;  (* Executa Grafcet *)
END_VAR
VAR_GLOBAL RETAIN
    G_550U1 : Grafcet550U1;
END_VAR
VAR_GLOBAL
    Exec_G_550U1 : BOOL;  (* Executa Grafcet *)
    TRG_530U1 : BOOL;  (* Trigger Leitor Código de Barras *)
    TRG_530U2 : BOOL;  (* Trigger Leitor Código de Barras *)
END_VAR
VAR_GLOBAL RETAIN
    G_540M1 : Grafcet540M1;
END_VAR
VAR_GLOBAL
    Zona530Auto : BOOL;  (* Zona em Automatico; published *)
    J02_EstbTargetSta : ARRAY[0..63] OF BOOL;  (* at IOBus://rack#0/slot#1/EstbTargetSta *)
    Exec_G_540M1 : BOOL;  (* Executa Grafcet *)
END_VAR
VAR_GLOBAL RETAIN
    G_610M1 : Grafcet6X0M1_Transport;
END_VAR
VAR_GLOBAL
    Zona540Auto : BOOL;  (* Zona em Automatico; published *)
    A_550U : AlarmeGeralEquipamento;  (* published *)
    Zona550Auto : BOOL;  (* Zona em Automatico; published *)
    I_550PS1 : BOOL;  (* 550PS1 - Botão Ok Impressora; at IOBus://rack#0/slot#3/Ch3_In/Ch3_In15 *)
    I_610YS2 : BOOL;
    Zona600Auto : BOOL;  (* Zona em Automatico; published *)
    Exec_G_610M1 : BOOL;  (* Executa Grafcet *)
END_VAR
VAR_GLOBAL RETAIN
    G_620M1 : Grafcet6X0M1_Transport;
END_VAR
VAR_GLOBAL
    I_620YS2 : BOOL;
    Exec_G_620M1 : BOOL;  (* Executa Grafcet *)
END_VAR
VAR_GLOBAL RETAIN
    G_630M1 : Grafcet6X0M1_Transport;
END_VAR
VAR_GLOBAL
    Exec_G_630M1 : BOOL;  (* Executa Grafcet *)
END_VAR
VAR_GLOBAL RETAIN
    G_640M1 : Grafcet6X0M1_Transport_Com2Transfer;
END_VAR
VAR_GLOBAL
    I_630YS2 : BOOL;
END_VAR
VAR_GLOBAL RETAIN
    G_640M2 : Grafcet6X0M1_Transport_Com2Transfer;
END_VAR
VAR_GLOBAL
    Exec_G_640M1 : BOOL;  (* Executa Grafcet *)
    I_641YS1 : BOOL;
    I_640YS2 : BOOL;
    I_641YS2 : BOOL;
    I_641XS1 : BOOL;
    I_641XS2 : BOOL;
    Exec_G_640M2 : BOOL;  (* Executa Grafcet *)
    I_642YS1 : BOOL;
    I_642YS2 : BOOL;
    I_643YS2 : BOOL;
    I_643YS1 : BOOL;
    I_642XS2 : BOOL;
    I_642XS1 : BOOL;
    I_643XS2 : BOOL;
    I_643XS1 : BOOL;
    SafetyIn : SafetyIn_struct;
    SafetyOut : SafetyOut_struct;
    A_020A1 : AlarmeGeralEquipamento;  (* published *)
    MachineID530M1 : UINT;  (* published *)
    MachineID540M1 : UINT;  (* published *)
    MachineID610M1 : UINT;  (* published *)
    MachineID620M1 : UINT;  (* published *)
    MachineID630M1 : UINT;  (* published *)
    MachineID640M1 : UINT;  (* published *)
    MachineID640M2 : UINT;  (* published *)
END_VAR

